# EPICS substitutions: fastFeedbackApp/Db/common/fbckIoc.substitutions
#==============================================================================
#
# Abs:  FBCK records for a single Feedback IOC
#
# Name: fbckIoc.substitutions
#
# Note: Must follow the LCLS naming conventions.
#
# NOTE: This file includes fbck records for the feedback IOCs
#       These records store function names of functions available on this ioc
#       modified:
#
# REVISION: (ababbitt) 2/19/2015 -  Updating the Macro substitution
#  to match this format  ("IOC_NAME",  "${IOC_TYPE}:${LOCA}:${LOOP}")
#
#==============================================================================
#
#
# ioc level config pvs
file fbckIocConfig.db {
	pattern {   IOC,     LC, LOOP, AREA }
	        { $(IOC),  $(LC), $(LP), $(AR) }
}
# ioc level status pvs
file fbckIocStatus.db {
	pattern {   IOC,     LC,  LOOP,  AREA }
	        { $(IOC),  $(LC), $(LP), $(AR) }
}
